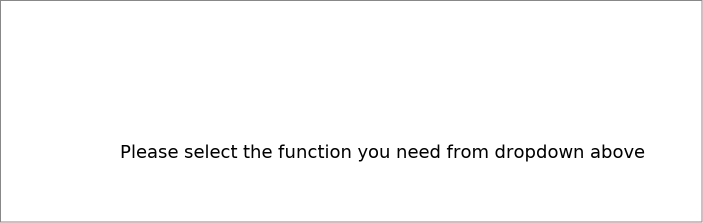
VISUALIZATION Visu_Welcome  // 703x223
    Rectangle (62,81 641x142), "Please select the function you need from dropdown above"
END_VISUALIZATION

(* stored: Version 1.1.0.1
   Visu Visu_Welcome: Id {cc543077-9835-49ce-9d3e-5a20695d1d9e} *)
